FUNCTION convertTimerToDisplayValue : INT
VAR_IN_OUT
	timerTon		:	TON;
END_VAR
VAR
END_VAR

convertTimerToDisplayValue := TIME_TO_INT ((GVL.configValues.minIdleSec - timerTon.ET) / 1000);

END_FUNCTION

(* stored: Version 1.1.0.1
   POU convertTimerToDisplayValue: Id {69bee498-1257-4038-bf88-af12297272dc}, SpecialFunc None *)
